// TIA Portal V20 export
TYPE "LConSMC_typeTechnologyControllerConfig"
// Konfiguration des Technologiereglers (Tänzer oder Zugmessdose) / Configuration parameters for technology controller (Dancer or load cell)
// stored: Access Published
   STRUCT
      x1 : LReal := 0.0;   // Stützpunkt 1 - X-Achse für P-Adaption (Wenn x1=x2 ist die Adaption deaktiviert) / Breakpoint 1 x-axis for P-adaption (if x1=x2 the adaption is deactivated)
      Kp1 : LReal := 1.0;   // Stützpunkt 1 - P-Verstärkung für P-Adaption (Wenn x1=x2 ist die Adaption deaktiviert) / Breakpoint 1 P-gain for P-adaption (if x1=x2 the adaption is deactivated)
      x2 : LReal;   // Stützpunkt 2 - X-Achse für P-Adaption (Wenn x1=x2 ist die Adaption deaktiviert) / Breakpoint 2 x-axis for P-adaption (if x1=x2 the adaption is deactivated)
      Kp2 : LReal := 1.0;   // Stützpunkt 2 - P-Verstärkung für P-Adaption (Wenn x1=x2 ist die Adaption deaktiviert) / Breakpoint 2 P-gain for P-adaption (if x1=x2 the adaption is deactivated)
      KpAdaptionValue : LReal := 0.0;   // Adaptionswert x-Achse für die Adaption der P-Verstärkung des Reglers / Adaption value for P-Gain adaption of the controller
      integTime : LReal := 2000.0;   // [ms] Integrationszeitkonstante Ein Wert von 0 deaktiviert den I-Anteil / [ms] Time constant for integrator. A value of 0 disables the I-part
      derivTime : LReal := 0.0;   // [ms] Differentationszeitkonstante Ein Wert von 0 deaktiviert den D-Anteil / [ms] Time constant for differentiator. A value of 0 disables the D-part
      derivControlMode : Bool := FALSE;   // TRUE: D-Komponente aktiv im Istwert-Pfad FALSE: D-Komponente aktiv in der Reglerabweichung / TRUE: D component active in actual value branch FALSE: D component in controller deviation
      setNominalValue : LReal := 100.0;   // Normierungswert für die Hochlaufzeit des Sollwertkanals (Rampen von 0 auf "setNominalValue" in "setRampTime") / Reference value for ramp time of setpoint channel (Ramp from 0 to "setNominalValue" in "setRampTime")
      setRampTime : LReal := 1000.0;   // [ms] Rampenzeit für Sollwertkanal / [ms] Ramp time for setpoint ramp generator
      filterTime : LReal := 10.0;   // [ms] PT1 - Istwertfilter Ein Wert von 0 deaktiviert den Filter / [ms] PT1- Filter for actual value. A value of 0 disables the filter
      intSetValue : LReal := 0.0;   // Setzwert des Integrators (wenn "setIntChannel" = TRUE) / Integrator set value (if "setIntChannel" = TRUE)
      setIntChannel : Bool := FALSE;   // TRUE: Der Wert des Integrators wird auf "intSetValue" gesetzt / TRUE: The output of the integrator is set to "intSetValue"
      holdIntChannel : Bool := FALSE;   // TRUE: Der Ausgang des Integrators wird gehalten FALSE: Der Integrator ist freigegeben / TRUE: The output of the integrator is hold FALSE: The output is integrated
      deadBand : LReal := 0.0;   // Breite des Totbandes (symmetrisch). Ein Wert von 0 deaktiviert das Totband / Value of the dead band (symmetrical). A value of 0 disables the deadband
      outValueFactor : LReal := 1.0;   // Multiplikativer Skalierungsfaktor des Reglerausgangs / Multiplicative scaling of the controller output
      upperLimit : LReal := 20.0;   // Oberer Grenze des Reglerausgangs / Upper limit of the controller output
      lowerLimit : LReal := -20.0;   // Untere Grenze des Reglerausgangs / Lower limit of the controller output
      limRampTime : LReal := 0.0;   // [ms] Hoch-/Rücklaufzeit für die Reglerausgangsbegrenzungen / [ms] Ramp time for output value limitation
      tensionReference : LReal := 0.0;   // [N oder lbf] Bezugswert für Zug-Sollwert Wenn der Wert 0 ist, wird der Sollwert als Absolutwert statt als Prozentwert interpretiert. / [N or lbf] Reference value for tension setpoint If the value is 0 the setpoint is interpreted as an abolute value and not percentage
   END_STRUCT;
END_TYPE
